// TIA Portal V21 export
TYPE "Std_eSavingResponse"
   STRUCT
      reserved { ExternalVisible := 'False'} : Int;
      saving_in_progress { ExternalVisible := 'False'} : Int := 1;
      saving_successful { ExternalVisible := 'False'} : Int := 2;
      saving_not_possible { ExternalVisible := 'False'} : Int := 3;
      saving_failed { ExternalVisible := 'False'} : Int := 4;
      access_denied_WebConfig { ExternalVisible := 'False'} : Int := 10;
      access_denied_saving { ExternalVisible := 'False'} : Int := 11;
      no_valve_detected { ExternalVisible := 'False'} : Int := 15;
      preparing_to_save { ExternalVisible := 'False'} : Int := 20;
      ready_to_save { ExternalVisible := 'False'} : Int := 21;
      FB_needs_rising_edge_xExecute { ExternalVisible := 'False'} : Int := 25;
   END_STRUCT;
END_TYPE
